GLOBALCONSTANTS HANDLE (* Global constants *)
  (* Standard: 61499-1 *)
  (* Version 1.0, 2025-09-04, franz *)
  PACKAGE isobus::pgn;
  VAR_GLOBAL CONSTANT
    UNVALID : INT := (-1);
    GLOBAL : INT := 32767; (* < \brief 0xFFFF Invalid or unused handle *)
  END_VAR
END_GLOBALCONSTANTS
